PROGRAM PRG_PID_CALL
VAR
	//B28
	B28_MTR_1_PID : PlantAndCMs.FB_PID;
	
	
END_VAR

(*
// MOTOR 1 PID CALL
HMI.CM_MTR_1_PID_PARAMS.tCtrlCycleTime := T#500MS;
HMI.CM_MTR_1_PID_PARAMS.tTaskCycleTime := T#100MS;
HMI.CM_MTR_1_PID_PARAMS.fKp := 5.0;	
HMI.CM_MTR_1_PID_PARAMS.tTd := T#500MS;
HMI.CM_MTR_1_PID_PARAMS.tTn := T#100S;
HMI.CM_MTR_1_PID_PARAMS.tTv := T#200MS;	
HMI.CM_MTR_1_PID_PARAMS.fOutMinLimit := 0.0;
HMI.CM_MTR_1_PID_PARAMS.fOutMaxLimit := 100.0;


B28_MTR_1_PID(
	IN_stCTRL_PID_PARAMS := HMI.CM_MTR_1_PID_PARAMS
	);

HMI.CM_DMP_1_PID_PARAMS.tCtrlCycleTime := T#500MS;
HMI.CM_DMP_1_PID_PARAMS.tTaskCycleTime := T#100MS;
HMI.CM_DMP_1_PID_PARAMS.fKp := 5.0;	
HMI.CM_DMP_1_PID_PARAMS.tTd := T#500MS;
HMI.CM_DMP_1_PID_PARAMS.tTn := T#100S;
HMI.CM_DMP_1_PID_PARAMS.tTv := T#200MS;	
HMI.CM_DMP_1_PID_PARAMS.fOutMinLimit := 0.0;
HMI.CM_DMP_1_PID_PARAMS.fOutMaxLimit := 180.0;

B28_DMP_1_PID(
	IN_stCTRL_PID_PARAMS := HMI.CM_MTR_1_PID_PARAMS
	);
*)

PRG_FB_CTRL_PID();

END_PROGRAM

(* stored: Version 1.1.0.1, ProductVersion 3.1.4024.13
   POU PRG_PID_CALL: Id {72632576-8a01-4602-b918-380b388b44b7}, SpecialFunc None *)
